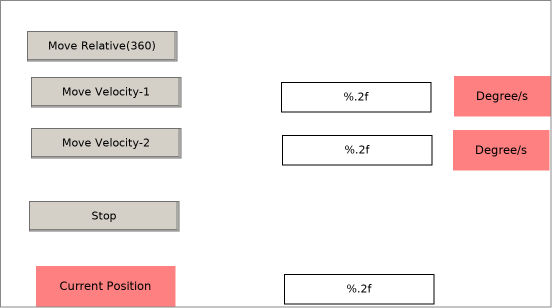
VISUALIZATION vis_motion  // 552x308
    Button (27,31 150x30), "Move Relative(360)"
        tap gHMI.bMoveRel
    Button (31,77 150x30), "Move Velocity-1"
        tap gHMI.bMoveVel
    Button (29,201 150x30), "Stop"
        tap gHMI.bStop
    Rectangle (453,130 96x40), "Degree/s"
    Rectangle (454,76 96x40), "Degree/s"
    Button (31,128 150x30), "Move Velocity-2"
        tap gHMI.bMoveVel2
    Rectangle (281,82 150x30), "%.2f", text variable: gHMI.vel
    Rectangle (282,135 150x30), "%.2f", text variable: gHMI.vel2
    Rectangle (36,266 139x40), "Current Position"
    Rectangle (284,274 150x30), "%.2f", text variable: gHMI.pos
END_VISUALIZATION

(* stored: Version 1.1.0.1, ProductVersion 3.1.4024.0
   Visu vis_motion: Id {3f34c172-c1f1-4f7a-ba0c-083ec4acc86b} *)
